FUNCTION_BLOCK FB_EmptyBlock
VAR_INPUT
END_VAR
VAR_OUTPUT
END_VAR
VAR
END_VAR

END_FUNCTION_BLOCK

(* stored: Version 1.1.0.1, ProductVersion 3.1.4024.12
   POU FB_EmptyBlock: Id {ff56077f-bb7b-4ae0-9c6e-4b14dcab3937}, SpecialFunc None *)
